TYPE Trapez :
STRUCT
	A	:REAL;
	B	:REAL;
	C	:REAL;
	D	:REAL;
END_STRUCT
END_TYPE

(* stored: Version 1.1.0.1, ProductVersion 3.1.4022.6
   DUT Trapez: Id {0b378636-8953-417e-9093-a4a3dac8387f} *)
